Omron CX-Programmer project NuevoProyecto (CX-Programmer 9.81)

# PLC NuevoPLC1: CPM2* 

## Global symbols (name address type ; comment)
0.00 BOOL  ; encendido
10.00 BOOL  ; verde
10.01 BOOL  ; AMARILLO
10.02 BOOL  ; ROJA

## Program NuevoPrograma1 (no task)

### Section Sección1

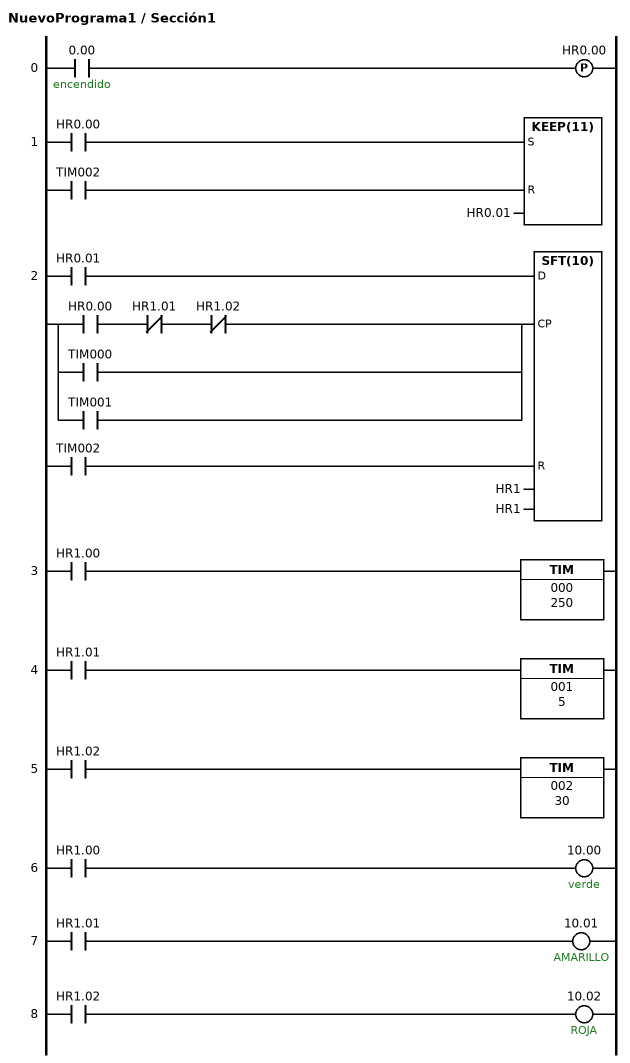
; rung 0
LD 0.00  ; encendido
DIFU(13) HR0.00
; rung 1
LD HR0.00
LD TIM002
KEEP(11) HR0.01
; rung 2
LD HR0.01
LD HR0.00
ANDNOT HR1.01
ANDNOT HR1.02
OR TIM000
OR TIM001
LD TIM002
SFT(10) HR1 HR1
; rung 3
LD HR1.00
TIM 000 250
; rung 4
LD HR1.01
TIM 001 5
; rung 5
LD HR1.02
TIM 002 30
; rung 6
LD HR1.00
OUT 10.00  ; verde
; rung 7
LD HR1.01
OUT 10.01  ; AMARILLO
; rung 8
LD HR1.02
OUT 10.02  ; ROJA

### Section END
; rung 0
END(01)